(* PLC project Unnamed, Unknown Unnamed 1 *)
(* stored: creationDateTime 2023-09-19T08:46:56, modificationDateTime 2023-12-05T13:42:59 *)

FUNCTION_BLOCK TP_WITH_RESET
  VAR_INPUT
    IN : BOOL;
    PT : TIME;
    RESET : BOOL;
  END_VAR
  VAR_OUTPUT
    Q : BOOL;
    ET : TIME := T#0s;
  END_VAR
  VAR
    STATE : SINT := 0;
    PREV_IN : BOOL := FALSE;
    CURRENT_TIME : TIME;
    START_TIME : TIME;
  END_VAR

            (* Pragma to set current time *)
{__SET_VAR(data__->,CURRENT_TIME,,__CURRENT_TIME)}

(*Timer block code *)
IF ((STATE = 0) AND NOT(PREV_IN) AND IN) THEN  (* found rising edge on IN *)
    (* start timer... *)
    STATE := 1;
    Q := TRUE;
    START_TIME := CURRENT_TIME;

ELSIF (STATE = 1) THEN (* timer counting *)
    IF ((START_TIME + PT) <= CURRENT_TIME) THEN (* timer expired *)
        STATE := 2;
        Q := FALSE;
        ET := PT;
    ELSE (* continue counting *)
        ET := CURRENT_TIME - START_TIME;
    END_IF;
END_IF;

IF ((STATE = 2) AND NOT(IN)) THEN
    ET := T#0s;
    STATE := 0;
END_IF;

IF (RESET) THEN (* reset pressed *)
  ET := T#0s;
  STATE := 0;
  Q := FALSE;
END_IF;

PREV_IN := IN;
          
END_FUNCTION_BLOCK

PROGRAM aplha
  VAR
    pwr_plant_switch AT %QX99.5 : BOOL;  (* Emergency cutoff *)
  END_VAR
  VAR
    pwr_plant : BOOL;
  END_VAR
  VAR
    pwr_gen AT %QX0.0 : BOOL;  (* Gen power on/ff *)
    pwr_buildings_on AT %QX0.1 : BOOL;  (* Defence estate power on *)
    pwr_buildings_off AT %QX0.2 : BOOL;  (* Defence estate power off *)
    pwr_hospital_on AT %QX0.3 : BOOL;  (* Field Hosp power on *)
    pwr_hospital_off AT %QX0.4 : BOOL;  (* Field Hosp power off *)
    alarm AT %QX0.5 : BOOL;  (* Power plant alarm *)
  END_VAR
  VAR
    alarm_start : BOOL;  (* Begin alarm loop *)
    alarm_reset : BOOL;  (* Continue alarm loop *)
    TP_WITH_RESET0 : TP_WITH_RESET;
    TP0 : TP;
  END_VAR
  VAR
    input_value_gen AT %QW0 : INT := 5000;  (* Generator HMI value *)
    input_value_pwr AT %QW1 : INT := 7000;  (* Power plant HMI value *)
    threshold_min_gen AT %QW2 : INT := 2000;  (* Generator low power threshold *)
    threshold_min_pwr AT %QW3 : INT := 5000;  (* Power plant low power threshold *)
  END_VAR
  VAR
    threshold_min_output_gen : BOOL;
    threshold_min_output_pwr : BOOL;
    CTU0 : CTU;
    temp_up : BOOL;
    temp_down : BOOL;
    max_temp : INT := 21;  (* Max temp value for vaccine serial *)
  END_VAR
  VAR
    current_temp AT %QW4 : INT;  (* Current temperature for vaccine storage *)
  END_VAR
  VAR
    temp_pulse : BOOL;
    TP2 : TP;
    TP_WITH_RESET1 : TP_WITH_RESET;
    temp_threshold : INT := 6;  (* Temp value at which temp alarm starts *)
  END_VAR
  VAR
    temp_alarm AT %QX99.4 : BOOL;  (* Initial temp alarm *)
    max_temp_alarm AT %QX99.7 : BOOL;  (* Max temp reached alarm *)
    gen_full AT %QW6 : INT := 100;  (* Set generator fuel to 100 *)
    fuel_value AT %QW5 : INT;  (* Current generator fuel value *)
  END_VAR
  VAR
    gen_empty : BOOL;
    gen_empty_pulse : BOOL;
    CTD0 : CTD;
    TP1 : TP;
    TP3 : TP;
  END_VAR
  VAR
    fuel_reset AT %QX99.6 : BOOL;
  END_VAR
  VAR
    max_pwr_plant : INT := 9000;  (* Max power threshold before power plant begins break cycle *)
  END_VAR
  VAR
    vape_smoke AT %QX0.7 : BOOL;  (* Smoke during break cycle *)
  END_VAR
  VAR
    TON0 : TON;
    pwr_plant_broke : BOOL;  (* Simulated break physical break of power plant *)
  END_VAR
  VAR  (* added by the conversion: wires and edge detectors of the diagram *)
    R_TRIG1 : R_TRIG;
    R_TRIG2 : R_TRIG;
  END_VAR

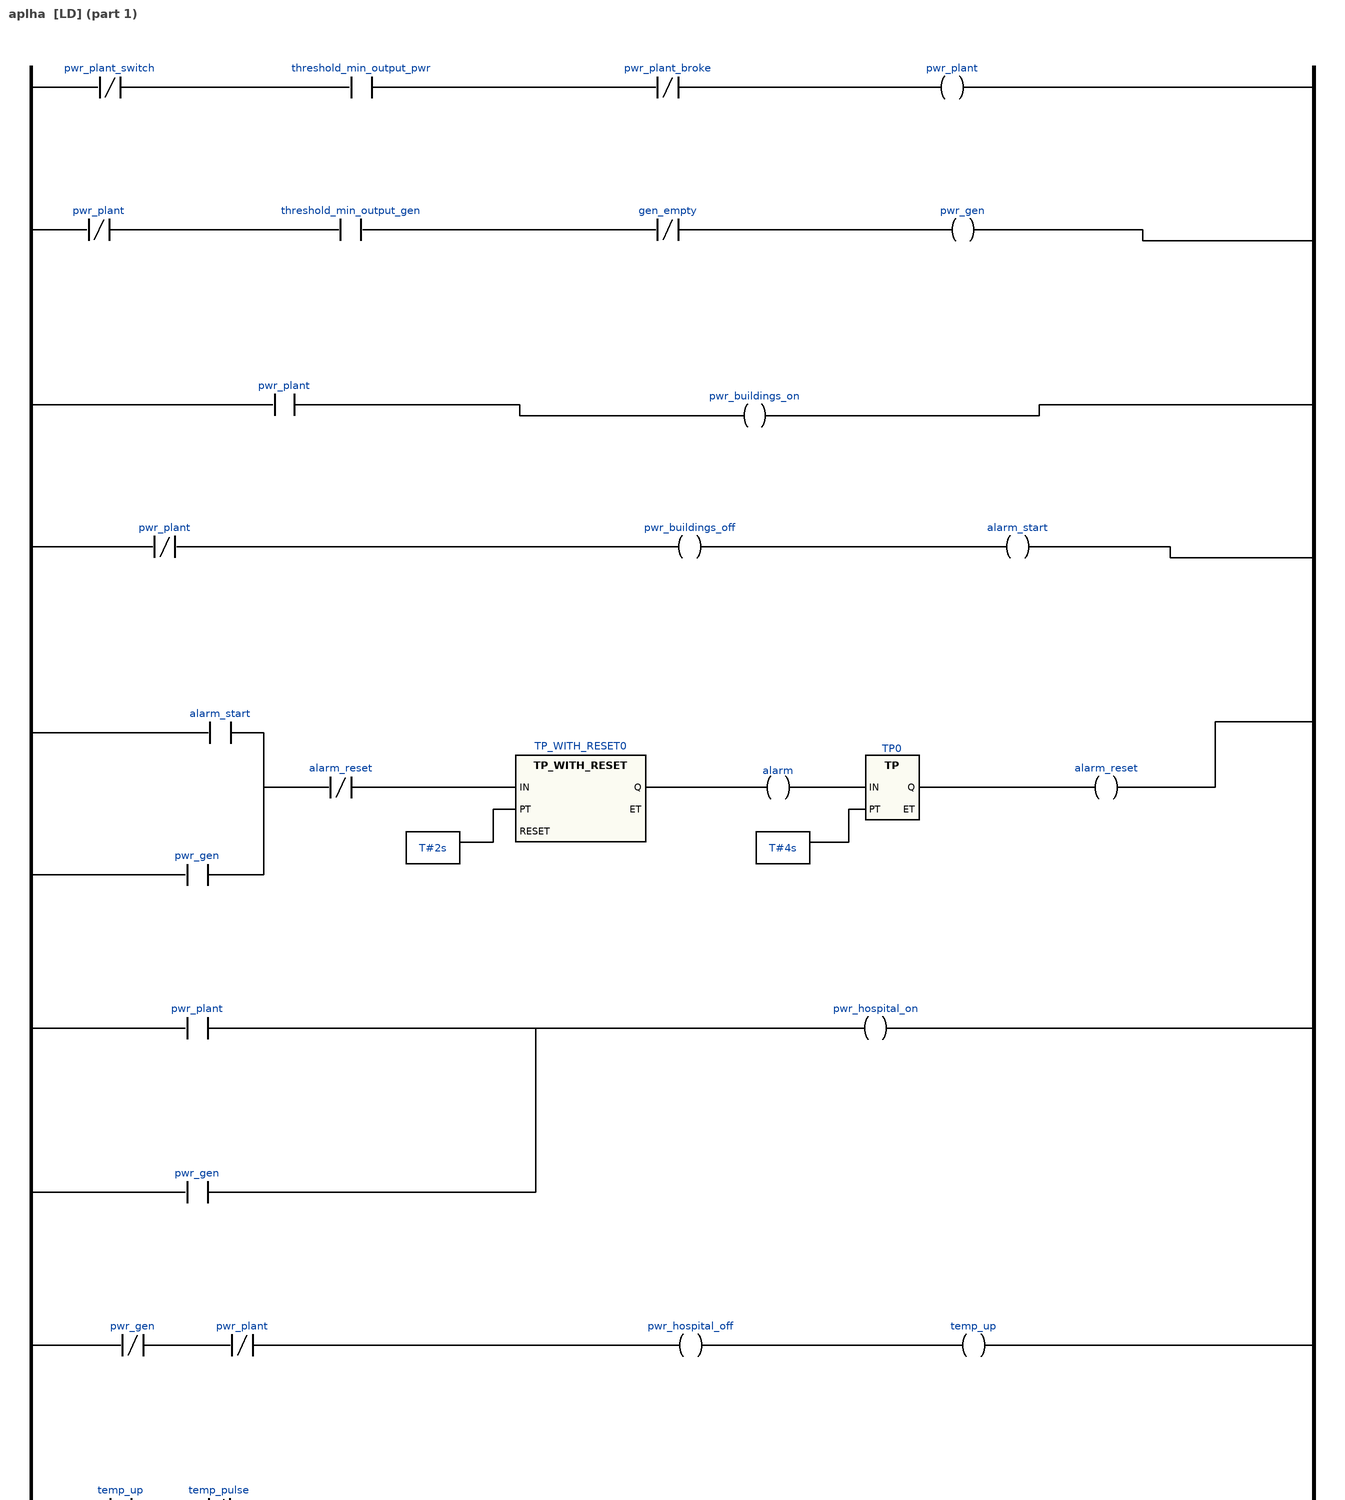
(* LD diagram, written out as Structured Text *)
pwr_plant := NOT pwr_plant_switch AND threshold_min_output_pwr AND NOT pwr_plant_broke;
pwr_gen := NOT pwr_plant AND threshold_min_output_gen AND NOT gen_empty;
pwr_buildings_on := pwr_plant;
pwr_buildings_off := NOT pwr_plant;
alarm_start := NOT pwr_plant;
TP_WITH_RESET0(IN := (alarm_start OR pwr_gen) AND NOT alarm_reset, PT := T#2s);
alarm := TP_WITH_RESET0.Q;
TP0(IN := TP_WITH_RESET0.Q, PT := T#4s);
alarm_reset := TP0.Q;
pwr_hospital_on := pwr_plant OR pwr_gen;
pwr_hospital_off := NOT pwr_gen AND NOT pwr_plant;
temp_up := NOT pwr_gen AND NOT pwr_plant;
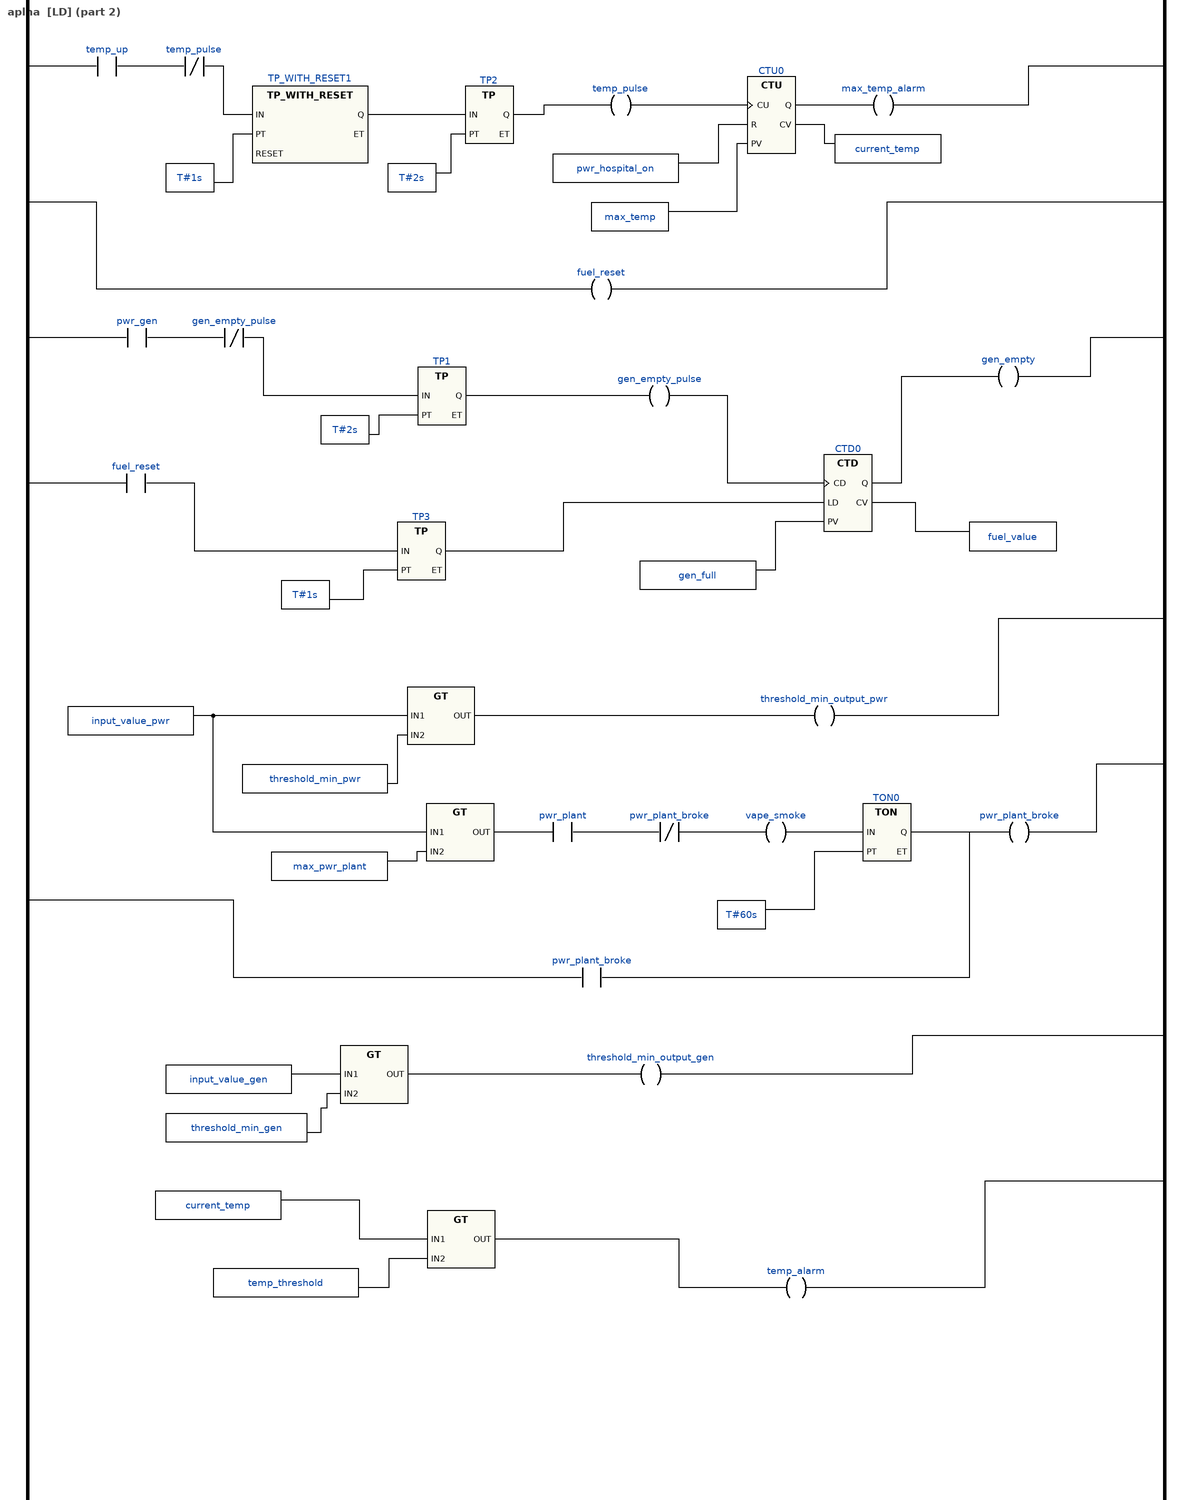
TP_WITH_RESET1(IN := temp_up AND NOT temp_pulse, PT := T#1s);
TP2(IN := TP_WITH_RESET1.Q, PT := T#2s);
temp_pulse := TP2.Q;
R_TRIG1(CLK := TP2.Q);
CTU0(CU := R_TRIG1.Q, R := pwr_hospital_on, PV := max_temp);
max_temp_alarm := CTU0.Q;
current_temp := CTU0.CV;
fuel_reset := TRUE;
TP1(IN := pwr_gen AND NOT gen_empty_pulse, PT := T#2s);
R_TRIG2(CLK := TP1.Q);
TP3(IN := fuel_reset, PT := T#1s);
CTD0(CD := R_TRIG2.Q, LD := TP3.Q, PV := gen_full);
gen_empty := CTD0.Q;
gen_empty_pulse := TP1.Q;
fuel_value := CTD0.CV;
threshold_min_output_pwr := input_value_pwr > threshold_min_pwr;
vape_smoke := input_value_pwr > max_pwr_plant AND pwr_plant AND NOT pwr_plant_broke;
TON0(IN := input_value_pwr > max_pwr_plant AND pwr_plant AND NOT pwr_plant_broke, PT := T#60s);
pwr_plant_broke := TON0.Q OR pwr_plant_broke;
threshold_min_output_gen := input_value_gen > threshold_min_gen;
temp_alarm := current_temp > temp_threshold;
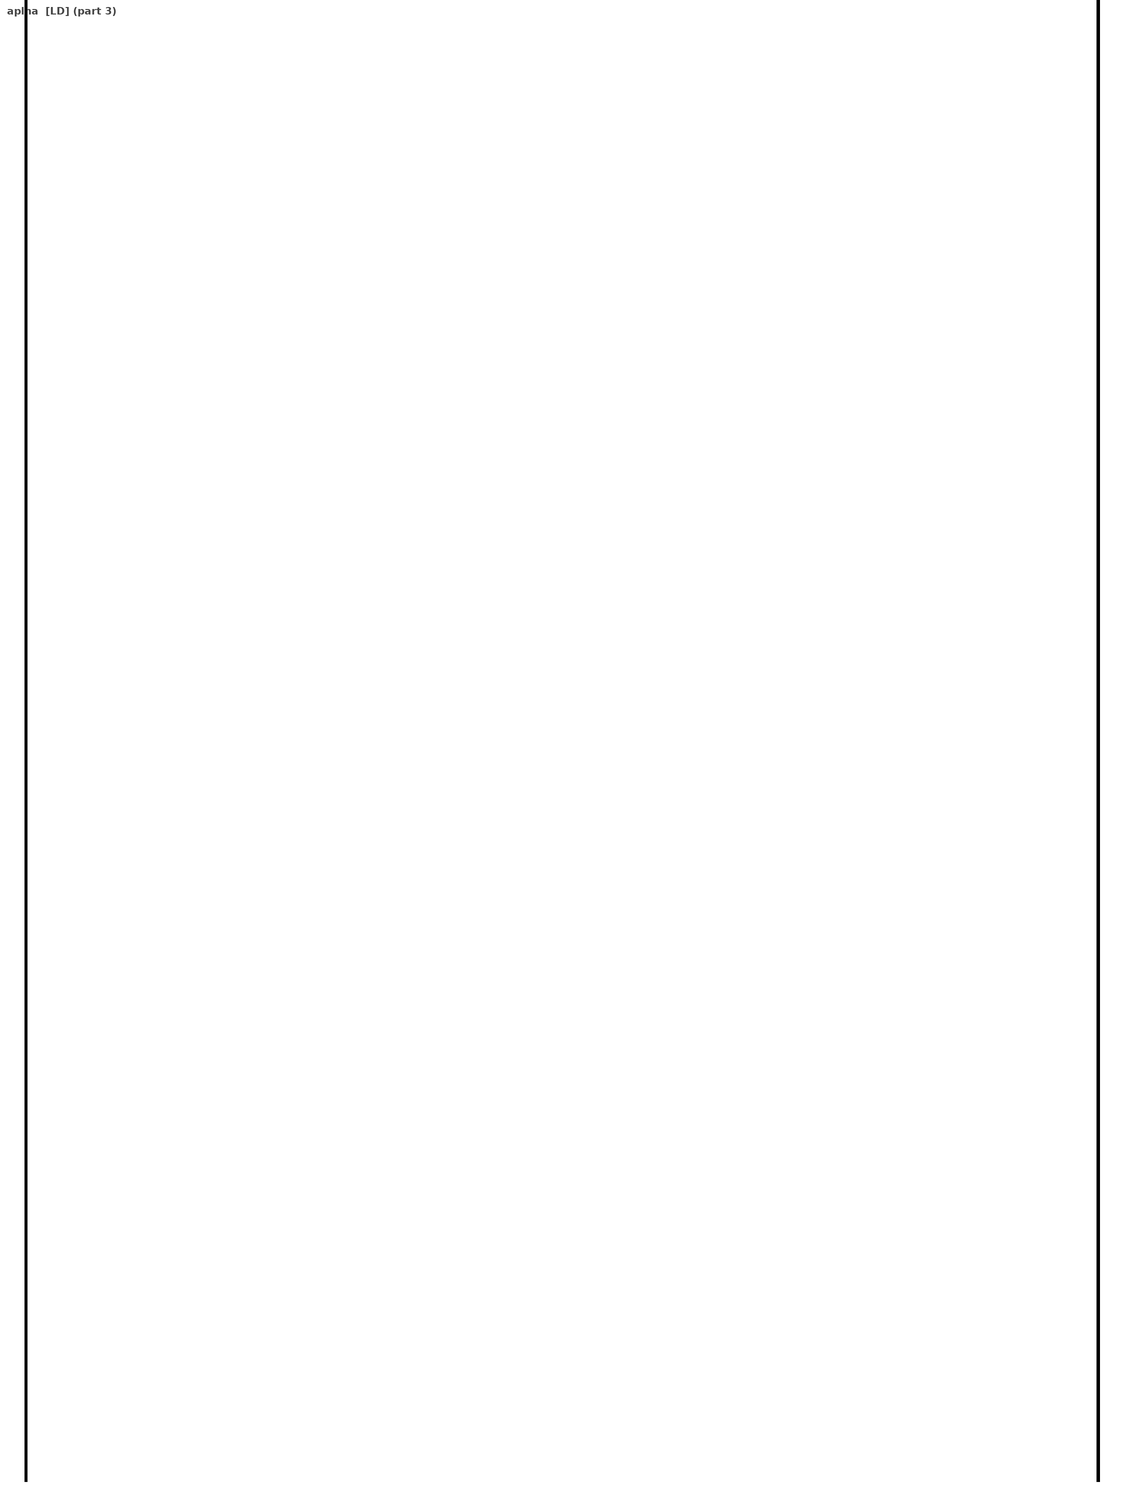
END_PROGRAM

CONFIGURATION Config0
  RESOURCE Res0 ON PLC
    TASK task0(INTERVAL := T#20ms, PRIORITY := 0);
    PROGRAM instance0 WITH task0 : aplha;
  END_RESOURCE
END_CONFIGURATION
